FUNCTION TryConvert_UDINT_TO_STRING : BOOL
VAR_INPUT
	in : UDINT;
	out : REFERENCE TO STRING;
END_VAR

out := UDINT_TO_STRING(in);
TryConvert_UDINT_TO_STRING := TRUE;

END_FUNCTION

(* stored: Version 1.1.0.1, ProductVersion 3.1.4024.12
   POU TryConvert_UDINT_TO_STRING: Id {51dc1576-1185-4e96-940c-2dc122fd4cdc}, SpecialFunc None *)
